{attribute 'qualified_only'}
TYPE E_PML_State :
(
    Undefined := 0,
    Stopped,
    Resetting,
    Idle,
    Starting,
    Execute,
    Completing,
    Complete,
    Holding,
    Held,
    Unholding,
    Stopping,
    Aborting,
    Aborted
) := Stopped;
END_TYPE

(* stored: Version 1.1.0.1, ProductVersion 3.1.4024.13
   DUT E_PML_State: Id {46620210-87b3-4e37-af63-cb8a280fcdb4} *)
